SUBAPPLICATION Uebung_006 (* Subapplication Type *)
  (* Standard: 61499-2 *)
  (* Version 1.0, 2023-10-23, franz *)
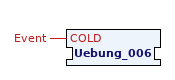
  EVENT_INPUT
    COLD;
  END_EVENT
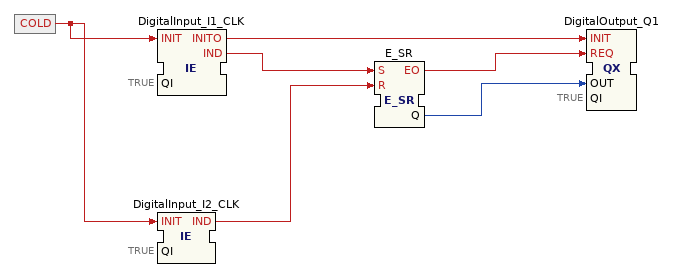
  FBS
    DigitalOutput_Q1 : QX(QI := TRUE);
    DigitalInput_I1_CLK : IE(QI := TRUE);
    DigitalInput_I2_CLK : IE(QI := TRUE);
    E_SR : E_SR;
  END_FBS
  EVENT_CONNECTIONS
    COLD TO DigitalInput_I1_CLK.INIT;
    DigitalInput_I1_CLK.INITO TO DigitalOutput_Q1.INIT;
    COLD TO DigitalInput_I2_CLK.INIT;
    DigitalInput_I1_CLK.IND TO E_SR.S;
    DigitalInput_I2_CLK.IND TO E_SR.R;
    E_SR.EO TO DigitalOutput_Q1.REQ;
  END_CONNECTIONS
  DATA_CONNECTIONS
    E_SR.Q TO DigitalOutput_Q1.OUT;
  END_CONNECTIONS
END_SUBAPPLICATION
